(* PLC project 01. MixingTank, CODESYS CODESYS V3.5 SP14 Patch 1, author Toni Kucic *)
(* stored: creationDateTime 2019-07-15T20:34:40.4571337, version 1.0, modificationDateTime 2019-07-15T20:34:40.3022281, organization TK Automation *)
(* This is a simulated mixing of two mediums in a tank. To see the full function description refer to the function description document. *)

PROGRAM MainProgram
  VAR
    Tank1FillingValveController : classFlipFlopCtrl;  (* ValveControllers *)
    Tank2FillingValveController : classFlipFlopCtrl;
    Tank3FillingValveController : classFlipFlopCtrl;
    Tank4FillingValveController : classFlipFlopCtrl;
    Tank1DrainValveController : classFlipFlopCtrl;
    Tank2DrainValveController : classFlipFlopCtrl;
    Tank3DrainValveController : classFlipFlopCtrl;
    Tank4DrainValveController : classFlipFlopCtrl;
    CollectionTankFillingValveController : classFlipFlopCtrl;
    CollectionTankDrainValveController : classFlipFlopCtrl;
    Tank1Control : TankControl;  (* Tank controllers *)
    Tank2Control : TankControl;
    Tank3Control : TankControl;
    Tank4Control : TankControl;
    CollectionTankControl : TankControl;
    Pump1Controller : classFlipFlopCtrl;  (* Pump controllers *)
    Pump2Controller : classFlipFlopCtrl;
    vRecirculationSP : REAL;  (* Support variables *)
    vNoOfFilling : REAL;
    vLevelRef : REAL;
    vFillingRef : REAL;
    vMaxTankLevel : REAL := 85;
    CollectingTankFillingValveOpene : INT;
  END_VAR
  VAR CONSTANT
    cTank1Capacity : REAL := 125;
    cTank2Capacity : REAL := 125;
    cTank3Capacity : REAL := 125;
    cTank4Capacity : REAL := 125;
    cMaxTankLevel : REAL := 80;
    cMinStorageTankLevel : REAL := 20;
  END_VAR

                    Pump1Controller(
	CloseAutoCmd := NOT IO.Pump1Running,
	OpenAutoCmd := NOT IO.CollectingTankDrainValveOpened OR IO.CollectingTankLevel_pc < 10,
	Opened := NOT IO.Pump1Running,
	Closed := IO.Pump1Running,
	qCloseCmd => IO.Pump1StartCmd,
	qOpenCmd => IO.Pump1StopCmd);

Pump2Controller(
	CloseAutoCmd := NOT IO.Pump2Running,
	OpenAutoCmd := NOT IO.CollectingTankDrainValveOpened OR IO.CollectingTankLevel_pc < 10,
	Opened := NOT IO.Pump2Running,
	Closed := IO.Pump2Running,
	qCloseCmd => IO.Pump2StartCmd,
	qOpenCmd => IO.Pump2StopCmd);
	
vLevelRef := ((0.01 * IO.Tank1Level_pc * cTank1Capacity 
		   + 0.01 * IO.Tank2Level_pc * cTank2Capacity 
		   + 0.01 * IO.Tank3Level_pc * cTank3Capacity 
		   + 0.01 * IO.Tank4Level_pc * cTank4Capacity)
		/(cTank1Capacity + cTank2Capacity + cTank3Capacity + cTank4Capacity));

vFillingRef := vMaxTankLevel - vLevelRef*100;

vNoOfFilling := BOOL_TO_REAL(IO.Tank1FillingValveOpened)
			+	BOOL_TO_REAL(IO.Tank2FillingValveOpened)
			+ 	BOOL_TO_REAL(IO.Tank3FillingValveOpened)
			+ 	BOOL_TO_REAL(IO.Tank4FillingValveOpened);	   
		   
Tank1Control(
	Tanklevel_pc := IO.Tank1Level_pc,
	LevelRef := vLevelRef * 100 + vFillingRef);
	
Tank2Control(
	Tanklevel_pc := IO.Tank2Level_pc,
	LevelRef := vLevelRef * 100 + vFillingRef);	

Tank3Control(
	Tanklevel_pc := IO.Tank3Level_pc,
	LevelRef := vLevelRef * 100 + vFillingRef);
	
Tank4Control(
	Tanklevel_pc := IO.Tank4Level_pc,
	LevelRef := vLevelRef * 100 + vFillingRef);
	
CollectionTankControl(
	Tanklevel_pc := IO.CollectingTankLevel_pc,
	LevelRef := IO.CollectingTankLevel_pc);
	
(* Commands to valves *)
Tank1FillingValveController(
	CloseAutoCmd := NOT Tank1Control.Fill,
	OpenAutoCmd := Tank1Control.Fill,
	Opened := IO.Tank1FillingValveOpened,
	Closed := IO.Tank1FillingValveClosed,
	qCloseCmd => IO.Tank1FillingValveCloseCmd,
	qOpenCmd => IO.Tank1FillingValveOpenCmd);
	
Tank2FillingValveController(
	CloseAutoCmd := NOT Tank2Control.Fill,
	OpenAutoCmd := Tank2Control.Fill,
	Opened := IO.Tank2FillingValveOpened,
	Closed := IO.Tank2FillingValveClosed,
	qCloseCmd => IO.Tank2FillingValveCloseCmd,
	qOpenCmd => IO.Tank2FillingValveOpenCmd);

Tank3FillingValveController(
	CloseAutoCmd := NOT Tank3Control.Fill,
	OpenAutoCmd := Tank3Control.Fill,
	Opened := IO.Tank3FillingValveOpened,
	Closed := IO.Tank3FillingValveClosed,
	qCloseCmd => IO.Tank3FillingValveCloseCmd,
	qOpenCmd => IO.Tank3FillingValveOpenCmd);
	
Tank4FillingValveController(
	CloseAutoCmd := NOT Tank4Control.Fill,
	OpenAutoCmd := Tank4Control.Fill,
	Opened := IO.Tank4FillingValveOpened,
	Closed := IO.Tank4FillingValveClosed,
	qCloseCmd => IO.Tank4FillingValveCloseCmd,
	qOpenCmd => IO.Tank4FillingValveOpenCmd);

Tank1DrainValveController(
	CloseAutoCmd := NOT Tank1Control.Drain,
	OpenAutoCmd := Tank1Control.Drain,
	Opened := IO.Tank1DrainValveOpened,
	Closed := IO.Tank1DrainValveClosed,
	qCloseCmd => IO.Tank1DrainValveCloseCmd,
	qOpenCmd => IO.Tank1DrainValveOpenCmd);
	
Tank2DrainValveController(
	CloseAutoCmd := NOT Tank2Control.Drain,
	OpenAutoCmd := Tank2Control.Drain,
	Opened := IO.Tank2DrainValveOpened,
	Closed := IO.Tank2DrainValveClosed,
	qCloseCmd => IO.Tank2DrainValveCloseCmd,
	qOpenCmd => IO.Tank2DrainValveOpenCmd);

Tank3DrainValveController(
	CloseAutoCmd := NOT Tank3Control.Drain,
	OpenAutoCmd := Tank3Control.Drain,
	Opened := IO.Tank3DrainValveOpened,
	Closed := IO.Tank3DrainValveClosed,
	qCloseCmd => IO.Tank3DrainValveCloseCmd,
	qOpenCmd => IO.Tank3DrainValveOpenCmd);
	
Tank4DrainValveController(
	CloseAutoCmd := NOT Tank4Control.Drain,
	OpenAutoCmd := Tank4Control.Drain,
	Opened := IO.Tank4DrainValveOpened,
	Closed := IO.Tank4DrainValveClosed,
	qCloseCmd => IO.Tank4DrainValveCloseCmd,
	qOpenCmd => IO.Tank4DrainValveOpenCmd);
	
CollectionTankDrainValveController(
	CloseAutoCmd := NOT CollectionTankControl.Fill,
	OpenAutoCmd := CollectionTankControl.Fill,
	Opened := IO.CollectingTankDrainValveOpened,
	Closed := IO.CollectingTankDrainValveClosed,
	qCloseCmd => IO.CollectingTankDrainValveCloseCmd,
	qOpenCmd => IO.CollectingTankDrainValveOpenCmd);
	
CollectionTankFillingValveController(
	CloseAutoCmd := NOT CollectionTankControl.Drain,
	OpenAutoCmd := CollectionTankControl.Drain,
	Opened := IO.CollectingTankFillingValveOpened,
	Closed := IO.CollectingTankFillingValveClosed,
	qCloseCmd => IO.CollectingTankFillingValveCloseCmd,
	qOpenCmd => IO.CollectingTankFillingValveOpenCmd);

	
vRecirculationSP := 100 - (25 * vNoOfFilling);

(* Set up the recirculation valve *)
IF IO.RecirculationValvePosition < vRecirculationSP THEN
	IO.OpenRecirculationValveCMD := TRUE;
	IO.CloseRecirculationValveCMD := FALSE;
ELSIF IO.RecirculationValvePosition > vRecirculationSP THEN
	IO.OpenRecirculationValveCMD := FALSE;
	IO.CloseRecirculationValveCMD := TRUE;
ELSE
	IO.OpenRecirculationValveCMD := FALSE;
	IO.CloseRecirculationValveCMD := FALSE;
END_IF
                  
END_PROGRAM

PROGRAM xsim01
  VAR
    Tank1 : Tank_Model;  (* Simulator and graphics Define objects *)
    Tank2 : Tank_Model;
    Tank3 : Tank_Model;
    Tank4 : Tank_Model;
    CollectingTank : Tank_Model;
    MapSignal : MapSignal;
    Pump1Sim : Pump_Model;
    Pump2Sim : Pump_Model;
    Tank1DrainValve : OnOffValve_model;
    Tank2DrainValve : OnOffValve_model;
    Tank3DrainValve : OnOffValve_model;
    Tank4DrainValve : OnOffValve_model;
    CollectingDrainValve : OnOffValve_model;
    Tank1FillingValve : OnOffValve_model;
    Tank2FillingValve : OnOffValve_model;
    Tank3FillingValve : OnOffValve_model;
    Tank4FillingValve : OnOffValve_model;
    CollectingFillingValve : OnOffValve_model;
    RecirculationValve : TwoWayIncrementValve;
    vPump1RunningDint : DINT;
    vPump2RunningDint : DINT;
    vPump1FlowRate : REAL;
    vPump2FlowRate : REAL;
    vCollectingTankName : STRING;
    vTank1Name : STRING;
    vTank1Nominal : INT;
    vTank2Nominal : INT;
    vTank2Name : STRING;
    vTank3Name : STRING;
    vTank3Nominal : INT;
    vTank4Name : STRING;
    vTank4Nominal : INT;
    vCollectingTankNom : INT;
    vCollectingTankLevel_cbm : REAL;
    vTank1Level_cbm : REAL;
    vTank4Level_cbm : REAL;
    vTank3Level_cbm : REAL;
    vTank2 : REAL;
    vTank2Level_cbm : REAL;
    vSystemFlowRate : REAL;
    vGravityDrain : REAL := 2500;
    vGravityFlowPerTank : INT;
    vNoOfDraining : DINT;
    vGravityDrainReturnFlow : REAL;
    vSystemFlowRatePerTank : REAL;
    vNoOfFilling : DINT;
    vReturnLineFlow : REAL;
    vSystemFlowRateTank1 : REAL;
    vSystemFlowRateTank2 : REAL;
    vSystemFlowRateTank3 : REAL;
    vSystemFlowRateTank4 : REAL;
    vGravityDrainTank1 : REAL;
    vGravityDrainTank2 : REAL;
    vGravityDrainTank3 : REAL;
    vGravityDrainTank4 : REAL;
    DischargeThreeWayValve : ThreeWayIncrementValve;
    vDischargedToOtherSystem : REAL;
    vThreeWayValvePos : REAL;
  END_VAR

                    (* Handle the valves *)
Tank1DrainValve(
	OpenCmd:= IO.Tank1DrainValveOpenCmd, 
	CloseCmd:= IO.Tank1DrainValveCloseCmd, 
	cfgOpeningTime:= T#3S, 
	cfgClosingTime:= T#3S, 
	simOpenFail:= FALSE, 
	simCloseFail:= FALSE, 
	Opened=> IO.Tank1DrainValveOpened, 
	Closed=> IO.Tank1DrainValveClosed );
	
Tank2DrainValve(
	OpenCmd:= IO.Tank2DrainValveOpenCmd, 
	CloseCmd:= IO.Tank2DrainValveCloseCmd, 
	cfgOpeningTime:= T#3S, 
	cfgClosingTime:= T#3S, 
	simOpenFail:= FALSE, 
	simCloseFail:= FALSE, 
	Opened=> IO.Tank2DrainValveOpened, 
	Closed=> IO.Tank2DrainValveClosed );

Tank3DrainValve(
	OpenCmd:= IO.Tank3DrainValveOpenCmd, 
	CloseCmd:= IO.Tank3DrainValveCloseCmd, 
	cfgOpeningTime:= T#3S, 
	cfgClosingTime:= T#3S, 
	simOpenFail:= FALSE, 
	simCloseFail:= FALSE, 
	Opened=> IO.Tank3DrainValveOpened, 
	Closed=> IO.Tank3DrainValveClosed );
	
Tank4DrainValve(
	OpenCmd:= IO.Tank4DrainValveOpenCmd, 
	CloseCmd:= IO.Tank4DrainValveCloseCmd, 
	cfgOpeningTime:= T#3S, 
	cfgClosingTime:= T#3S, 
	simOpenFail:= FALSE, 
	simCloseFail:= FALSE, 
	Opened=> IO.Tank4DrainValveOpened, 
	Closed=> IO.Tank4DrainValveClosed );
	
CollectingDrainValve(
	OpenCmd:= IO.CollectingTankDrainValveOpenCmd, 
	CloseCmd:= IO.CollectingTankDrainValveCloseCmd, 
	cfgOpeningTime:= T#3S, 
	cfgClosingTime:= T#3S, 
	simOpenFail:= FALSE, 
	simCloseFail:= FALSE, 
	Opened=> IO.CollectingTankDrainValveOpened, 
	Closed=> IO.CollectingTankDrainValveClosed );

Tank1FillingValve(
	OpenCmd:= IO.Tank1FillingValveOpenCmd, 
	CloseCmd:= IO.Tank1FillingValveCloseCmd, 
	cfgOpeningTime:= T#3S, 
	cfgClosingTime:= T#3S, 
	simOpenFail:= FALSE, 
	simCloseFail:= FALSE, 
	Opened=> IO.Tank1FillingValveOpened, 
	Closed=> IO.Tank1FillingValveClosed );
	
Tank2FillingValve(
	OpenCmd:= IO.Tank2FillingValveOpenCmd, 
	CloseCmd:= IO.Tank2FillingValveCloseCmd, 
	cfgOpeningTime:= T#3S, 
	cfgClosingTime:= T#3S, 
	simOpenFail:= FALSE, 
	simCloseFail:= FALSE, 
	Opened=> IO.Tank2FillingValveOpened, 
	Closed=> IO.Tank2FillingValveClosed );

Tank3FillingValve(
	OpenCmd:= IO.Tank3FillingValveOpenCmd, 
	CloseCmd:= IO.Tank3FillingValveCloseCmd, 
	cfgOpeningTime:= T#3S, 
	cfgClosingTime:= T#3S, 
	simOpenFail:= FALSE, 
	simCloseFail:= FALSE, 
	Opened=> IO.Tank3FillingValveOpened, 
	Closed=> IO.Tank3FillingValveClosed );
	
Tank4FillingValve(
	OpenCmd:= IO.Tank4FillingValveOpenCmd, 
	CloseCmd:= IO.Tank4FillingValveCloseCmd, 
	cfgOpeningTime:= T#3S, 
	cfgClosingTime:= T#3S, 
	simOpenFail:= FALSE, 
	simCloseFail:= FALSE, 
	Opened=> IO.Tank4FillingValveOpened, 
	Closed=> IO.Tank4FillingValveClosed );
	
CollectingFillingValve(
	OpenCmd:= IO.CollectingTankFillingValveOpenCmd, 
	CloseCmd:= IO.CollectingTankFillingValveCloseCmd, 
	cfgOpeningTime:= T#3S, 
	cfgClosingTime:= T#3S, 
	simOpenFail:= FALSE, 
	simCloseFail:= FALSE, 
	Opened=> IO.CollectingTankFillingValveOpened, 
	Closed=> IO.CollectingTankFillingValveClosed );
	
RecirculationValve(
	OpenCMD := IO.OpenRecirculationValveCMD,
	CloseCMD := IO.CloseRecirculationValveCMD,
	cfgTaskSeq_ms := 20,
	cfgOpenSpeed_s := 5,
	cfgCloseSpeed_s:= 5,
	Position => IO.RecirculationValvePosition);
	
DischargeThreeWayValve(
	ForwardCMD:= IO.DischargeThreeWayFwdCmd, 
	BackwardCMD:= IO.DischargeThreeWayBackCmd, 
	cfgTaskSeq_ms:= 20, 
	cfgOpenSpeed_s:= 5, 
	cfgCloseSpeed_s:= 5, 
	Position=> IO.DischargeThreeWayValvePosition );
	
(* Calculate the system values *)
vNoOfDraining := BOOL_TO_DINT(Tank1DrainValve.Opened)
				+ BOOL_TO_DINT(Tank2DrainValve.Opened)
				+ BOOL_TO_DINT(Tank3DrainValve.Opened)
				+ BOOL_TO_DINT(Tank4DrainValve.Opened);

vNoOfFilling := BOOL_TO_DINT(Tank1FillingValve.Opened)
				+ BOOL_TO_DINT(Tank2FillingValve.Opened)
				+ BOOL_TO_DINT(Tank3FillingValve.Opened)
				+ BOOL_TO_DINT(Tank4FillingValve.Opened);				
(* Handle the pumps *)
Pump1Sim(
	OnCmd:= IO.Pump1StartCmd, 
	OffCmd:= IO.Pump1StopCmd, 
	cfgFlowrate:= 2400,
	SimTrip:= IO.Pump1Running AND RecirculationValve.Position = 0 AND vNoOfFilling = 0,
	NoWater := CollectingTank.TankLevel_cbm = 0 OR CollectingDrainValve.Closed, 
	RunStatus=> vPump1RunningDint, 
	FlowmeterOut=> vPump1FlowRate);
	IO.Pump1Running:= DINT_TO_BOOL(vPump1RunningDint);
	
Pump2Sim(
	OnCmd:= IO.Pump2StartCmd, 
	OffCmd:= IO.Pump2StopCmd, 
	cfgFlowrate:= 2400,
	SimTrip:= IO.Pump2Running AND RecirculationValve.Position = 0 AND vNoOfFilling = 0,
	NoWater := CollectingTank.TankLevel_cbm = 0 OR CollectingDrainValve.Closed,  
	RunStatus=> vPump2RunningDint, 
	FlowmeterOut=> vPump2FlowRate);
	IO.Pump2Running:= DINT_TO_BOOL(vPump2RunningDint);
				
vSystemFlowRate := vPump1FlowRate + vPump2Flowrate;
vSystemFlowRateTank1 := 0.01*(100-RecirculationValve.Position)*(vSystemFlowRate / DINT_TO_REAL(MAX(1,vNoOfFilling))) * BOOL_TO_REAL(Tank1FillingValve.Opened);
vSystemFlowRateTank2 := 0.01*(100-RecirculationValve.Position)*(vSystemFlowRate / DINT_TO_REAL(MAX(1,vNoOfFilling))) * BOOL_TO_REAL(Tank2FillingValve.Opened);
vSystemFlowRateTank3 := 0.01*(100-RecirculationValve.Position)*(vSystemFlowRate / DINT_TO_REAL(MAX(1,vNoOfFilling))) * BOOL_TO_REAL(Tank3FillingValve.Opened);
vSystemFlowRateTank4 := 0.01*(100-RecirculationValve.Position)*(vSystemFlowRate / DINT_TO_REAL(MAX(1,vNoOfFilling))) * BOOL_TO_REAL(Tank4FillingValve.Opened);
vReturnLineFlow := vSystemFlowRate - vSystemFlowRateTank1 - vSystemFlowRateTank2 - vSystemFlowRateTank3 - vSystemFlowRateTank4;

IF IO.DischargeThreeWayValvePosition >= -45 AND IO.DischargeThreeWayValvePosition <= 90 THEN
	MapSignal(x1 := 0, x2 := 1, a1 := -45, a2 := 90, A := IO.DischargeThreeWayValvePosition, X => vThreeWayValvePos);
ELSIF IO.DischargeThreeWayValvePosition > 90 THEN
	MapSignal(x1 := 1, x2 := 0, a1 := 90, a2 := 180, A := IO.DischargeThreeWayValvePosition, X => vThreeWayValvePos);
END_IF;

vGravityDrainTank1 := (vGravityDrain / DINT_TO_REAL(MAX(1,vNoOfDraining)))* BOOL_TO_REAL(Tank1DrainValve.Opened AND Tank1.TankLevel_pc > 0);
vGravityDrainTank2 := (vGravityDrain / DINT_TO_REAL(MAX(1,vNoOfDraining)))* BOOL_TO_REAL(Tank2DrainValve.Opened AND Tank2.TankLevel_pc > 0);
vGravityDrainTank3 := (vGravityDrain / DINT_TO_REAL(MAX(1,vNoOfDraining)))* BOOL_TO_REAL(Tank3DrainValve.Opened AND Tank3.TankLevel_pc > 0);
vGravityDrainTank4 := (vGravityDrain / DINT_TO_REAL(MAX(1,vNoOfDraining)))* BOOL_TO_REAL(Tank4DrainValve.Opened AND Tank4.TankLevel_pc > 0);
//Dischargin possible from -10 to +180
// Gravity possible from -180 to 10
vDischargedToOtherSystem := (vGravityDrainTank1 +	vGravityDrainTank2 + vGravityDrainTank3 + vGravityDrainTank4) * LIMIT(0,vThreeWayValvePos, 1);
vGravityDrainReturnFlow := vGravityDrainTank1 +	vGravityDrainTank2 + vGravityDrainTank3 + vGravityDrainTank4 - vDischargedToOtherSystem;

Tank1(
	cfgTaskCycle:= 20, 
	cfgLenght:= 10, 
	cfgWidth:= 10, 
	cfgHeight:= 5, 
	cfgStartLevel:= 0, 
	Inflow1:= vSystemFlowRateTank1,
	Outflow1:= vGravityDrainTank1,
	TankLevel_cbm=>vTank1Level_cbm,
	TankLevel_pc=> IO.Tank1Level_pc);
	vTank1Name := 'Storage Tank 1';
	vTank1Nominal := 500;

Tank2(
	cfgTaskCycle:= 20, 
	cfgLenght:= 5, 
	cfgWidth:= 5, 
	cfgHeight:= 5, 
	cfgStartLevel:= 100, 
	Inflow1:= vSystemFlowRateTank2, 
	Outflow1:= vGravityDrainTank2,
	TankLevel_cbm=>vTank2Level_cbm,
	TankLevel_pc=> IO.Tank2Level_pc);
	vTank2Name := 'Storage Tank 2';
	vTank2Nominal := 125;
	
Tank3(
	cfgTaskCycle:= 20, 
	cfgLenght:= 5, 
	cfgWidth:= 5, 
	cfgHeight:= 5, 
	cfgStartLevel:= 100, 
	Inflow1:= vSystemFlowRateTank3, 
	Outflow1:= vGravityDrainTank3,
	TankLevel_cbm=>vTank3Level_cbm,
	TankLevel_pc=> IO.Tank3Level_pc);
	vTank3Name := 'Storage Tank 3';
	vTank3Nominal := 125;
	
Tank4(
	cfgTaskCycle:= 20, 
	cfgLenght:= 10, 
	cfgWidth:= 10, 
	cfgHeight:= 5, 
	cfgStartLevel:= 0, 
	Inflow1:= vSystemFlowRateTank4, 
	Outflow1:= vGravityDrainTank4,
	TankLevel_cbm=>vTank4Level_cbm,
	TankLevel_pc=> IO.Tank4Level_pc);
	vTank4Name := 'Storage Tank 4';
	vTank4Nominal := 500;

CollectingTank(
	cfgTaskCycle:= 20, 
	cfgLenght:= 10, 
	cfgWidth:= 10, 
	cfgHeight:= 10, 
	cfgStartLevel:= 333, 
	Inflow1:= 5000 * BOOL_TO_REAL(CollectingFillingValve.Opened), 
	Inflow2:= vGravityDrainReturnFlow,
	Inflow3:= vReturnLineFlow,
	Outflow1:= vSystemFlowRate * BOOL_TO_REAL(CollectingDrainValve.Opened),
	TankLevel_cbm=>vCollectingTankLevel_cbm,
	TankLevel_pc=> IO.CollectingTankLevel_pc);
	vCollectingTankName := 'Collecting Tank';
	vCollectingTankNom := 1000;

                  
END_PROGRAM

FUNCTION_BLOCK classFlipFlopCtrl
  VAR_INPUT
    SetAutoCmd : BOOL := FALSE;
    SetManCmd : BOOL := FALSE;
    CloseManCmd : BOOL := FALSE;
    OpenManCmd : BOOL := FALSE;
    CloseAutoCmd : BOOL := FALSE;
    OpenAutoCmd : BOOL := FALSE;
    Opened : BOOL := FALSE;
    Closed : BOOL := FALSE;
  END_VAR
  VAR_OUTPUT
    qCloseCmd : BOOL := FALSE;
    qOpenCmd : BOOL := FALSE;
  END_VAR
  VAR
    vSetAutoCmdOld : BOOL;
    vControlPos : INT := 0;
    vSetManCmdOld : BOOL;
    vErrorStateActive : BOOL;
  END_VAR

                    // Determine control position
IF (vControlPos = 0) AND SetAutoCmd AND NOT vSetAutoCmdOld THEN
	vControlPos := 1;
END_IF
IF (vControlPos = 1) AND SetManCmd AND NOT vSetManCmdOld THEN
	vControlPos := 0;
END_IF

IF vErrorStateActive THEN
	vControlPos := 0;
END_IF

CASE vControlPos OF
	0: (* Manual *)
	qCloseCmd := CloseManCmd AND NOT Closed;
	qOpenCmd := OpenManCmd AND NOT Opened;
	
	1: (* Auto *)
	qCloseCmd := CloseAutoCmd AND NOT Closed;
	qOpenCmd := OpenAutoCmd AND NOT Opened;
END_CASE

// Memory
vSetAutoCmdOld := SetAutoCmd;
vSetManCmdOld :=  SetManCmd;
                  
END_FUNCTION_BLOCK

PROGRAM ValveLogic
  VAR
    ON : BOOL;
    TripSeverity : INT;
    Voltage : INT := 110;
  END_VAR

                    ON := TripSeverity = 1 AND Voltage <= 100 OR ON AND TripSeverity = 1;

                  
END_PROGRAM

PROGRAM TankLogic

                    
                  
END_PROGRAM

FUNCTION_BLOCK MapSignal
  VAR_INPUT
    x1 : REAL;  (* Minimum range of output signal *)
    x2 : REAL;  (* Maximum range of output signal *)
    a1 : REAL;  (* Minimum range of input signal *)
    a2 : REAL;  (* Maximum range of input signal *)
    A : REAL;  (* Actual input signal *)
  END_VAR
  VAR_OUTPUT
    X : REAL;  (* Actual output signal *)
  END_VAR

                     X := (x2 - x1)*(A - a1)/(a2 - a1) + x1;
                  
END_FUNCTION_BLOCK

CONFIGURATION SoftPLC
  RESOURCE Application ON PLC
    {attribute 'qualified_only'}
    VAR_GLOBAL  (* IO *)
      Pump1StartCmd : BOOL;  (* DIGITAL OUTPUT Naredba automatike za start pumpe 1 *)
      Pump1StopCmd : BOOL;  (* DIGITAL OUTPUT Naredba automatike za stop pumpe 1 *)
      Pump1Running : BOOL;  (* DIGITAL INPUT Indikacija pokrenutog status pumpe 1 *)
      Pump2StartCmd : BOOL;  (* DIGITAL OUTPUT Naredba automatike za start pumpe 2 *)
      Pump2StopCmd : BOOL;  (* DIGITAL OUTPUT Naredba automatike za stop pumpe 2 *)
      Pump2Running : BOOL;  (* DIGITAL INPUT Indikacija pokrenutog status pumpe 2 *)
      Tank1Level_pc : REAL;  (* REAL VALUE Trenutna razina tanka u postocima *)
      Tank2Level_pc : REAL;  (* REAL VALUE Trenutna razina tanka u postocima *)
      Tank3Level_pc : REAL;  (* REAL VALUE Trenutna razina tanka u postocima *)
      Tank4Level_pc : REAL;  (* REAL VALUE Trenutna razina tanka u postocima *)
      CollectingTankLevel_pc : REAL;  (* REAL VALUE Trenutna razina tanka u postocima *)
      Tank1DrainValveOpenCmd : BOOL;
      Tank1DrainValveCloseCmd : BOOL;
      Tank1DrainValveOpened : BOOL;
      Tank1DrainValveClosed : BOOL;
      Tank2DrainValveOpenCmd : BOOL;
      Tank2DrainValveCloseCmd : BOOL;
      Tank2DrainValveOpened : BOOL;
      Tank2DrainValveClosed : BOOL;
      Tank3DrainValveOpenCmd : BOOL;
      Tank3DrainValveCloseCmd : BOOL;
      Tank3DrainValveOpened : BOOL;
      Tank3DrainValveClosed : BOOL;
      Tank4DrainValveOpenCmd : BOOL;
      Tank4DrainValveCloseCmd : BOOL;
      Tank4DrainValveOpened : BOOL;
      Tank4DrainValveClosed : BOOL;
      CollectingTankDrainValveOpenCmd : BOOL;
      CollectingTankDrainValveCloseCmd : BOOL;
      CollectingTankDrainValveOpened : BOOL;
      CollectingTankDrainValveClosed : BOOL;
      Tank1FillingValveOpenCmd : BOOL;
      Tank1FillingValveCloseCmd : BOOL;
      Tank1FillingValveOpened : BOOL;
      Tank1FillingValveClosed : BOOL;
      Tank2FillingValveOpenCmd : BOOL;
      Tank2FillingValveCloseCmd : BOOL;
      Tank2FillingValveOpened : BOOL;
      Tank2FillingValveClosed : BOOL;
      Tank3FillingValveOpenCmd : BOOL;
      Tank3FillingValveCloseCmd : BOOL;
      Tank3FillingValveOpened : BOOL;
      Tank3FillingValveClosed : BOOL;
      Tank4FillingValveOpenCmd : BOOL;
      Tank4FillingValveCloseCmd : BOOL;
      Tank4FillingValveOpened : BOOL;
      Tank4FillingValveClosed : BOOL;
      CollectingTankFillingValveOpenCmd : BOOL;
      CollectingTankFillingValveCloseCmd : BOOL;
      CollectingTankFillingValveOpened : BOOL;
      CollectingTankFillingValveClosed : BOOL;
      OpenRecirculationValveCMD : BOOL;
      CloseRecirculationValveCMD : BOOL;
      RecirculationValvePosition : REAL;
      DischargeThreeWayFwdCmd : BOOL;
      DischargeThreeWayBackCmd : BOOL;
      DischargeThreeWayValvePosition : REAL;
    END_VAR
    TASK xsim01(INTERVAL := T#20ms, PRIORITY := 1);
    TASK VISU_TASK(INTERVAL := T#50ms, PRIORITY := 31);
    TASK xc01_Task(INTERVAL := T#50ms, PRIORITY := 1);
    PROGRAM xsim01 WITH xsim01 : xsim01;
    PROGRAM VisuElems.Visu_Prg WITH VISU_TASK : VisuElems.Visu_Prg;
    PROGRAM MainProgram WITH xc01_Task : MainProgram;
    PROGRAM ValveLogic WITH xc01_Task : ValveLogic;
  END_RESOURCE
END_CONFIGURATION
